INTERFACE I_NodePrototypes

METHOD PUBLIC Accept
VAR_INPUT
	Visitor : I_NodePrototypeVisitor;
END_VAR
END_METHOD

END_INTERFACE

(* stored: Version 1.1.0.1, ProductVersion 3.1.4024.12
   Itf I_NodePrototypes: Id {f17dfa9a-d58a-0253-28a9-a9333d414dc7}
   Method Accept: Id {130c651f-9790-4ffb-80fd-ac3f957fad9e} *)
